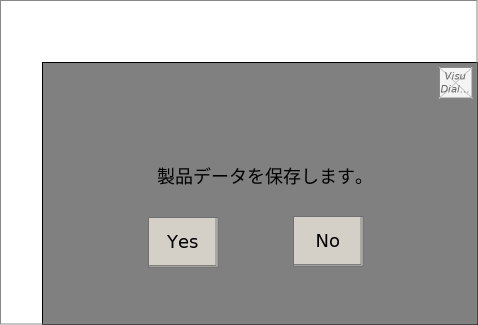
VISUALIZATION d_saveProduct  // 478x325
    Rectangle (42,62 436x263)
    Image (439,67 33x31), image: VisuDialogs.ImagePoolDialogs.Delete
        OnMouseClick: CloseDialog Dialog=d_saveProduct, Result=OK, NumpadKeypadSet=True
    Label (69,146 392x62), "製品データを保存します。"
    Button (148,217 70x50), "Yes"
        tap gvl_visu.flg_btn_saveProductInfo
        OnMouseClick: CloseDialog Dialog=d_saveProduct, Result=OK, NumpadKeypadSet=True
    Button (293,216 70x50), "No"
        OnMouseClick: CloseDialog Dialog=d_saveProduct, Result=OK, NumpadKeypadSet=True
END_VISUALIZATION

(* stored: Version 1.1.0.1, ProductVersion 3.1.4024.12
   Visu d_saveProduct: Id {a79ce421-735e-42fb-aa17-62ee0193752f} *)
